{attribute addProperty BoxType "EPP1321-0060-0016"}
{attribute addProperty Id "A_0019_EPP1322_0001_0016A_0019_EPP1322_0001_0016_1D2305932662332.75"}
{attribute addProperty CRC "3479285291"}
{attribute addProperty SizeInBites "2662"}
{attribute addProperty SizeInBytes "332.75"}
TYPE A_0018_EPP1321_0060_0016_CF61AE2B EXTENDS EPP1321_179A0949 :
STRUCT
	{attribute addProperty Name "A_0019_EPP1322_0001_0016"}
	A_0019_EPP1322_0001_0016 : A_0019_EPP1322_0001_0016_1D230593;
END_STRUCT
END_TYPE

(* stored: Version 1.2.0.0, ProductVersion 3.1.4024.9
   DUT A_0018_EPP1321_0060_0016_CF61AE2B: Id {0d2f51e0-6d25-40c2-b119-ef27aac3322c} *)
